TYPE ST_Parameters_PRR :
STRUCT
	methodName		: STRING;
	revision		: DINT;
	createdBy		: STRING;
	createdDate		: STRING;
	solv_R1			: DINT;
	solv_R2			: DINT;
	solv_W1			: DINT;
	solv_W2			: DINT;
	stepTime_R1		: DINT;
	stepTime_R2		: DINT;
	stepTime_W1		: DINT;
	stepTime_W2		: DINT;
	stepRpm_R1		: DINT;
	stepRpm_R2		: DINT;
	stepRpm_W1		: DINT;
	stepRpm_W2		: DINT;
	soakTime		: DINT;
	agitateTime1	: DINT;
	agitateTime2	: DINT;
	vialToFill		: DINT;
	vialPrimeVol	: REAL;
	vialFillVol1	: REAL;
	vialsFillVol24	: REAL;
	airDryTime		: DINT;
END_STRUCT
END_TYPE

(* stored: Version 1.1.0.1, ProductVersion 3.1.4024.12
   DUT ST_Parameters_PRR: Id {90a7c414-4e14-4ca4-8a58-cfe0b7a3981a} *)
